FUNCTION_BLOCK AX_TLIM (* Standard timer function block (time-limiting, timeout) *)
  (* Standard: 61499-2; Classification: standard timer function block; Description: Copyright (c) 2026 HR Agrartechnik GmbH This program and the accompanying materials are made available under the terms of the Eclipse Public License 2.0 which is available at https://www.eclipse.org/legal/epl-2.0/ SPDX-License-Identifier: EPL-2.0 AX_TLIM -- Time-limiting timer FB with AX adapter interface The adapter input IN triggers execution (E1->REQ) and provides the boolean input value (D1->IN). The event input EIPT presets the time limit PT without triggering execution. When IN goes TRUE, Q becomes TRUE and a timer starts. If IN stays TRUE longer than PT, Q goes FALSE (timeout). If IN goes FALSE before PT expires, Q goes FALSE immediately. *)
  (* Version 1.0, 2026-05-08, Franz Höpfinger, HR Agrartechnik GmbH, initial API and implementation and/or initial documentation *)
  PACKAGE adapter::events::unidirectional::timers;
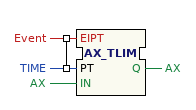
  EVENT_INPUT
    EIPT WITH PT; (* Set Preset Time (non-triggering) *)
  END_EVENT
  VAR_INPUT
    PT : TIME; (* Time limit *)
  END_VAR
  SOCKETS
    IN : adapter::types::unidirectional::AX; (* Timer input (AX adapter) *)
  END_SOCKETS
  PLUGS
    Q : adapter::types::unidirectional::AX; (* Timer output (AX adapter) *)
  END_PLUGS
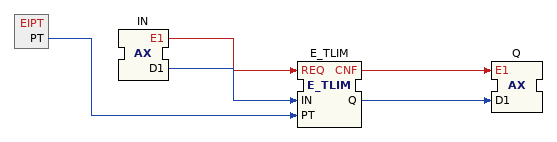
  FBS
    E_TLIM : iec61499::events::timers::E_TLIM;
  END_FBS
  EVENT_CONNECTIONS
    E_TLIM.CNF TO Q.E1;
    IN.E1 TO E_TLIM.REQ;
  END_CONNECTIONS
  DATA_CONNECTIONS
    E_TLIM.Q TO Q.D1;
    IN.D1 TO E_TLIM.IN;
    PT TO E_TLIM.PT;
  END_CONNECTIONS
END_FUNCTION_BLOCK
